% RSLogix 500 project PLC-Controlled Simulated Pick-and-Place System with E-Stop & Loop Mode.RSS, saved by version 8.30.00.16 %
PROJECT "UNTITLED"    % processor: Bul.1763 MicroLogix 1100 Series B %

PROGRAM FILES
  LAD 2 "MAIN"  9 rungs
  LAD 3 "SAFETY"  4 rungs
  LAD 4 "MODES"  4 rungs

DATA FILES
  O0 OUTPUT  4 elements
  I1 INPUT  6 elements
  S2 STATUS  66 elements
  B3 BINARY  10 elements
  T4 TIMER  3 elements
  C5 COUNTER  1 elements
  R6 CONTROL  1 elements
  N7 INTEGER  1 elements
  F8 FLOAT  1 elements

LADDER 2 "MAIN"
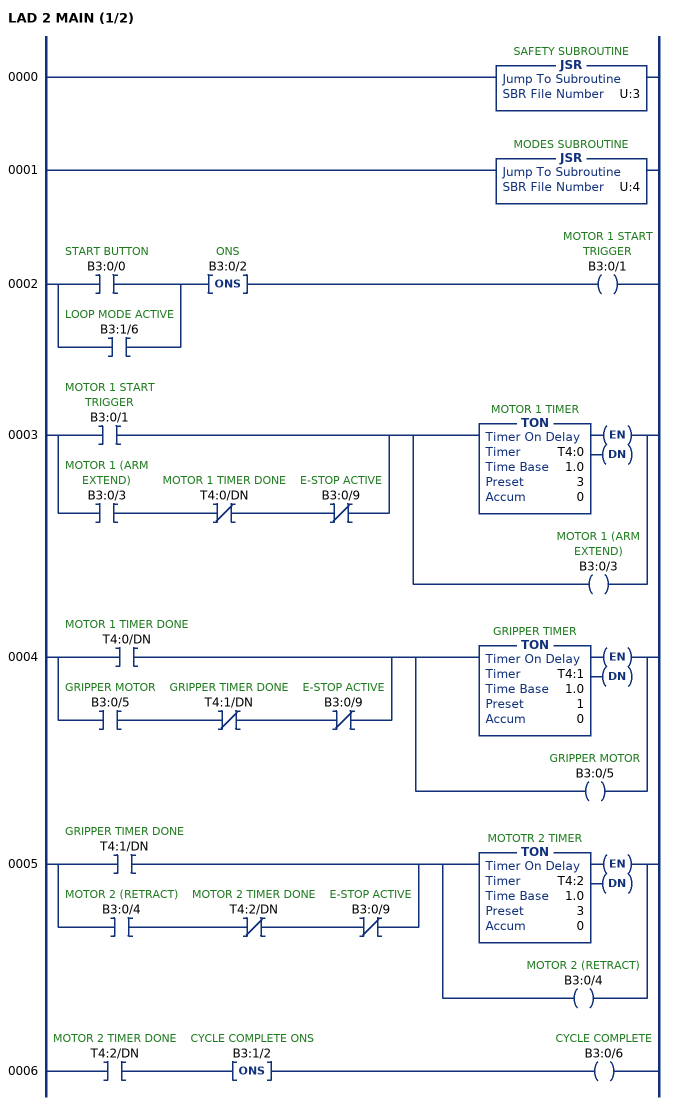
% Rung: 0 %
SOR JSR U:3 EOR
%   U:3  "SAFETY SUBROUTINE" %
% Rung: 1 %
SOR JSR U:4 EOR
%   U:4  "MODES SUBROUTINE" %
% Rung: 2 %
SOR BST XIC B3:0/0 NXB XIC B3:1/6 BND ONS B3:0/2 OTE B3:0/1 EOR
%   B3:0/0  "START BUTTON" %
%   B3:1/6  "LOOP MODE ACTIVE" %
%   B3:0/2  "ONS" %
%   B3:0/1  "MOTOR 1 START TRIGGER" %
% Rung: 3 %
SOR BST XIC B3:0/1 NXB XIC B3:0/3 XIO T4:0/DN XIO B3:0/9 BND BST TON T4:0 1.0 3 0 NXB OTE B3:0/3 BND EOR
%   B3:0/1  "MOTOR 1 START TRIGGER" %
%   B3:0/3  "MOTOR 1 (ARM EXTEND)" %
%   T4:0/DN  "MOTOR 1 TIMER DONE" %
%   B3:0/9  "E-STOP ACTIVE" %
%   T4:0  "MOTOR 1 TIMER" %
% Rung: 4 %
SOR BST XIC T4:0/DN NXB XIC B3:0/5 XIO T4:1/DN XIO B3:0/9 BND BST TON T4:1 1.0 1 0 NXB OTE B3:0/5 BND EOR
%   T4:0/DN  "MOTOR 1 TIMER DONE" %
%   B3:0/5  "GRIPPER MOTOR" %
%   T4:1/DN  "GRIPPER TIMER DONE" %
%   B3:0/9  "E-STOP ACTIVE" %
%   T4:1  "GRIPPER TIMER" %
% Rung: 5 %
SOR BST XIC T4:1/DN NXB XIC B3:0/4 XIO T4:2/DN XIO B3:0/9 BND BST TON T4:2 1.0 3 0 NXB OTE B3:0/4 BND EOR
%   T4:1/DN  "GRIPPER TIMER DONE" %
%   B3:0/4  "MOTOR 2 (RETRACT)" %
%   T4:2/DN  "MOTOR 2 TIMER DONE" %
%   B3:0/9  "E-STOP ACTIVE" %
%   T4:2  "MOTOTR 2 TIMER" %
% Rung: 6 %
SOR XIC T4:2/DN ONS B3:1/2 OTE B3:0/6 EOR
%   T4:2/DN  "MOTOR 2 TIMER DONE" %
%   B3:1/2  "CYCLE COMPLETE ONS" %
%   B3:0/6  "CYCLE COMPLETE" %

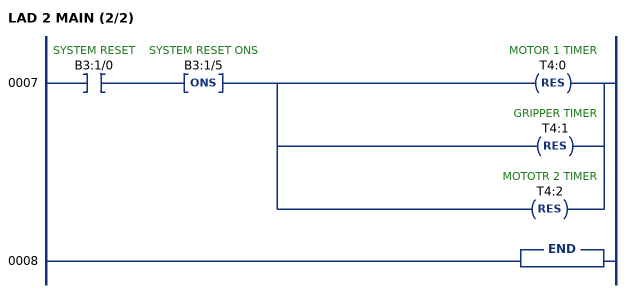
% Rung: 7 %
SOR XIC B3:1/0 ONS B3:1/5 BST RES T4:0 NXB RES T4:1 NXB RES T4:2 BND EOR
%   B3:1/0  "SYSTEM RESET" %
%   B3:1/5  "SYSTEM RESET ONS" %
%   T4:0  "MOTOR 1 TIMER" %
%   T4:1  "GRIPPER TIMER" %
%   T4:2  "MOTOTR 2 TIMER" %
% Rung: 8 %
SOR END EOR

LADDER 3 "SAFETY"
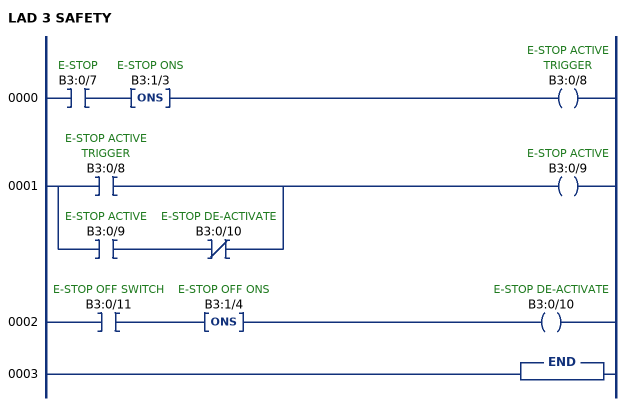
% Rung: 0 %
SOR XIC B3:0/7 ONS B3:1/3 OTE B3:0/8 EOR
%   B3:0/7  "E-STOP" %
%   B3:1/3  "E-STOP ONS" %
%   B3:0/8  "E-STOP ACTIVE TRIGGER" %
% Rung: 1 %
SOR BST XIC B3:0/8 NXB XIC B3:0/9 XIO B3:0/10 BND OTE B3:0/9 EOR
%   B3:0/8  "E-STOP ACTIVE TRIGGER" %
%   B3:0/9  "E-STOP ACTIVE" %
%   B3:0/10  "E-STOP DE-ACTIVATE" %
% Rung: 2 %
SOR XIC B3:0/11 ONS B3:1/4 OTE B3:0/10 EOR
%   B3:0/11  "E-STOP OFF SWITCH" %
%   B3:1/4  "E-STOP OFF ONS" %
%   B3:0/10  "E-STOP DE-ACTIVATE" %
% Rung: 3 %
SOR END EOR

LADDER 4 "MODES"
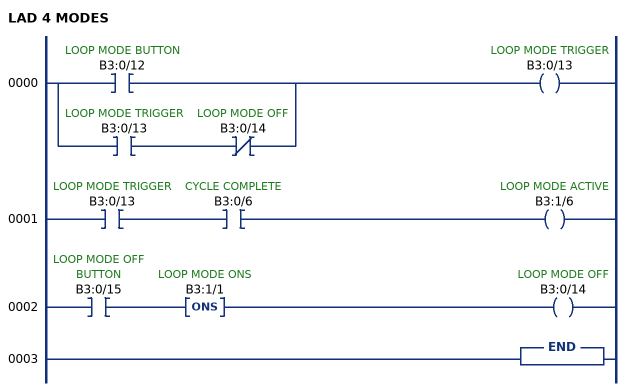
% Rung: 0 %
SOR BST XIC B3:0/12 NXB XIC B3:0/13 XIO B3:0/14 BND OTE B3:0/13 EOR
%   B3:0/12  "LOOP MODE BUTTON" %
%   B3:0/13  "LOOP MODE TRIGGER" %
%   B3:0/14  "LOOP MODE OFF" %
% Rung: 1 %
SOR XIC B3:0/13 XIC B3:0/6 OTE B3:1/6 EOR
%   B3:0/13  "LOOP MODE TRIGGER" %
%   B3:0/6  "CYCLE COMPLETE" %
%   B3:1/6  "LOOP MODE ACTIVE" %
% Rung: 2 %
SOR XIC B3:0/15 ONS B3:1/1 OTE B3:0/14 EOR
%   B3:0/15  "LOOP MODE OFF BUTTON" %
%   B3:1/1  "LOOP MODE ONS" %
%   B3:0/14  "LOOP MODE OFF" %
% Rung: 3 %
SOR END EOR

DATA TABLE (non-zero values as saved)
DATA T4
% .PRE .ACC %
% T4:0 % 3 0
% T4:1 % 1 0
% T4:2 % 3 0
